// TIA Portal V17 export
// export: Created 2026-04-13T11:12:44.9223065Z, ExportSetting WithDefaults, DisplayName Totally Integrated Automation Portal, DisplayVersion V17 Update 4, DisplayName TIA Portal Openness, DisplayVersion V17 Update 4, DisplayName TIA Portal Version Control Interface, DisplayVersion V17, DisplayName SINAMICS Startdrive Advanced, DisplayVersion V17, DisplayName SINAMICS Startdrive G130, G150, S120, S150, SINAMICS MV, S210, DisplayVersion V17, DisplayName SINAMICS Startdrive G110M, G120, G120C, G120D, G120P, G115D, DisplayVersion V17, DisplayName STEP 7 Professional, DisplayVersion V17 Update 4, DisplayName STEP 7 Safety, DisplayVersion V17, DisplayName WinCC Professional, DisplayVersion V17 Update 4
FUNCTION_BLOCK "Modbus_Master"   // FB641, SCL
TITLE = Modbus master communication
AUTHOR : SIMATIC
FAMILY : MODBUS
NAME : MB_MASTR
VERSION : 5.0
// stored: IsIECCheckEnabled true, SetENOAutomatically false, UDAEnableTagReadback false
   VAR_INPUT
      REQ : Bool;   // Startet die angeforderte Übertragung bei steigender Flanke / Activates the requested transmission on rising edge
      MB_ADDR : UInt;   // Modbus RTU Stationsadresse / Modbus RTU station address
      MODE : USInt;   // Bezeichnet die Art der Anforderung / Specifies the type of request
      DATA_ADDR : UDInt;   // Anfangsadresse im Slave / Starting Address in the Slave
      DATA_LEN : UInt;   // Datenlänge: Anzahl der Bits oder Wörter / Specifies the number of bits or words to be accessed
   END_VAR
   VAR_OUTPUT
      DONE : Bool;   // Anweisung beendet ohne Fehler / Instruction finished without error
      BUSY : Bool;   // Modbus Master Auftrag in Arbeit / Modbus master transaction in progress
      ERROR : Bool;   // Anweisung beendet mit Fehler / Instruction finished with error
      STATUS : Word := 16#7000;   // Detailllierte Fehlerinformation / Detailed error information
   END_VAR
   VAR_IN_OUT
      DATA_PTR : Variant;   // Referenz auf die lokale Quell- oder Zieladresse / Reference to the local source or destination address
   END_VAR
   VAR DB_SPECIFIC
      MB_State : SInt := 0;   // Internal state of the Modbus master operation
      Blocked_Proc_Timeout : Real := 3.0;   // Time to wait upon a blocked Modbus Master instance before setting inactive
      Extended_Addressing : Bool;   // Configures slave addressing; 1=double-byte adressing
      Compatibility_Mode : Bool;   // 1= data transfer for FC1, FC2 and FC15 compatible with CP341
      MB_DB { S7_SetPoint := 'True'} : P2P_MB_BASE;   // Modbus parameters
   END_VAR
   VAR
      Send_P2P { S7_SetPoint := 'True'} : Send_P2P;   // Local instance of the instruction Send_P2P
      Receive_P2P { S7_SetPoint := 'True'} : Receive_P2P;   // Local instance of the instruction Receive_P2P
      Receive_Reset { S7_SetPoint := 'True'} : Receive_Reset;   // Local instance of the instruction Receive_Reset
   END_VAR
   VAR DB_SPECIFIC
      S_PORT : Word;   // For internal use only
      S_RESP_TO : Word;   // For internal use only
      S_ICHAR_GAP : Word;   // For internal use only
      S_RETRIES : Word;   // For internal use only
      S_MB_ADDR : UInt;   // Modbus RTU station address
      S_MODE : USInt;   // Specifies the type of request
      S_DATA_ADDR : UDInt;   // Starting Address in the Slave
      S_DATA_LEN : UInt;   // Specifies the number of bits or words to be accessed
      w_retries : Word;   // For internal use only
      y_SlaveAddrHi : Byte;   // For internal use only
      y_SlaveAddrLo : Byte;   // For internal use only
      StartAddress : Word;   // For internal use only
      Value : Word;   // For internal use only
      y_FCode : Byte;   // For internal use only
   END_VAR
   VAR
      FCode_usint AT y_FCode : USInt;
   END_VAR
   VAR DB_SPECIFIC
      INTERNAL_CDATA : Array[1..257] of Byte;   // For internal use only
   END_VAR
   VAR
      FC1_2_Req AT INTERNAL_CDATA : P2P_MB_FC1_2_Req;   // For internal use only
      FC1_4_ValResp AT INTERNAL_CDATA : P2P_MB_FC1_4_ValResp;   // For internal use only
      FC3_4_Req AT INTERNAL_CDATA : P2P_MB_FC3_4_Req;   // For internal use only
      FC5_6_Req AT INTERNAL_CDATA : P2P_MB_FC5_6_Req;   // For internal use only
      FC5_6_ValResp AT INTERNAL_CDATA : P2P_MB_FC5_6_ValResp;   // For internal use only
      FC15_16_Req AT INTERNAL_CDATA : P2P_MB_FC15_16_Req;   // For internal use only
      FC11_Req AT INTERNAL_CDATA : P2P_MB_FC11_Req;   // For internal use only
      FC11_ValResp AT INTERNAL_CDATA : P2P_MB_FC11_ValResp;   // For internal use only
      FC8_Req AT INTERNAL_CDATA : P2P_MB_FC8_Req;   // For internal use only
      FCx_ErrResp AT INTERNAL_CDATA : P2P_MB_FCx_ErrResp;   // For internal use only
      MB_Header AT INTERNAL_CDATA : Struct
         free : Byte;
         SlaveAddrHi : Byte;
         SlaveAddrLo : Byte;
         FCode : Byte;
         addr : UInt;
         quantity_value : UInt;
      END_STRUCT;
      FC11 AT INTERNAL_CDATA : Struct
         free : Byte;
         SlaveAddrHi : Byte;
         SlaveAddrLo : Byte;
         FCode : Byte;
         data : Array[0..3] of Byte;
      END_STRUCT;
   END_VAR
   VAR DB_SPECIFIC
      mb_timer { S7_SetPoint := 'True'} : TON_TIME;
      TimeElapsed : Bool;
   END_VAR
BEGIN
END_FUNCTION_BLOCK
